{attribute 'linkalways'} 
{attribute 'no_explicit_call' := 'This FB is a CLASS and must be accessed using methods or properties'}
{attribute 'enable_dynamic_creation'}
FUNCTION_BLOCK FINAL GE_LINT EXTENDS Node
VAR
	in1 : _LINT(0);
	in2 : _LINT(0);
	out : _BOOL(FALSE);
END_VAR

METHOD PUBLIC Clone : I_Node
VAR
	pNode : POINTER TO GE_LINT;
END_VAR
pNode := __NEW(GE_LINT);
Clone := pNode^;
END_METHOD

METHOD FB_init : BOOL
VAR_INPUT
	bInitRetains : BOOL; // if TRUE, the retain variables are initialized (warm start / cold start)
	bInCopyCode : BOOL;  // if TRUE, the instance afterwards gets moved into the copy code (online change)
END_VAR
AddInput('in1',THIS^.in1);
AddInput('in2',THIS^.in2);
AddOutput('out', THIS^.out);
END_METHOD

METHOD PROTECTED OnExecute
VAR
END_VAR
out.Value := in1.Value >= in2.Value;
END_METHOD

END_FUNCTION_BLOCK

(* stored: Version 1.1.0.1, ProductVersion 3.1.4024.15
   POU GE_LINT: Id {3615acb2-fcc7-4ca8-bbaa-5d47cbbe3d41}, SpecialFunc None
   Folder Constructor: Id {d52625c5-2596-4f48-9b4b-48958e67f011}
   Method Clone: Id {ea833ff3-8b85-41a8-bea0-6738d2f87134}
   Method FB_init: Id {c9812adb-6831-476e-b6f5-18eaeaf4e7dc}
   Method OnExecute: Id {98f36f2c-3ae7-449d-b24f-1383f9cb6f90} *)
